{attribute 'qualified_only'}
VAR_GLOBAL
	//master_Ramp_Enable                   : BOOL;
	//master_Ramp_Value                    : ARRAY[1..4] OF LREAL;
	master_TargetTemp                    : LREAL;
	master_PowLimit_                     : ARRAY[1..4] OF LREAL;
	master_integral_constant			 : ARRAY[1..4] OF LREAL;	//PI제어기 적분상수
	master_pi_gain                       : ARRAY[1..4] OF LREAL;	//PI제어기 이득(gain)
	master_Sampling_Time				 : LREAL;  //Δt(*고정값*)
	master_Zone_Temp_Min_per             : LREAL;  //단위 : %
	master_Zone_Temp_Max_per             : LREAL;  //단위 : %
	master_fMV_Out						 : ARRAY[1..4] OF LREAL;
	
	master_tuning_mode 	     			 : BOOL;
	master_tuning_time	     			 : TIME;
	master_bWatch						 : BOOL;
END_VAR

(* stored: Version 1.1.0.1, ProductVersion 3.1.4024.4
   GVL mgbl: Id {76f52044-44fa-4847-aa89-50cabd58f1fc} *)
